// TIA Portal V17 export
BLOCK "F-FB_EStop"   // ObjectSW123, F-LAD
// failsafe emergency stop
// stored: IsFailsafe true
BEGIN

REGION Network 1: failsafe coil
END_REGION
END_BLOCK
